ABB RobotStudio station: Session3b.rspag

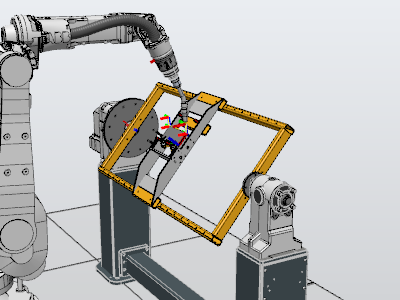
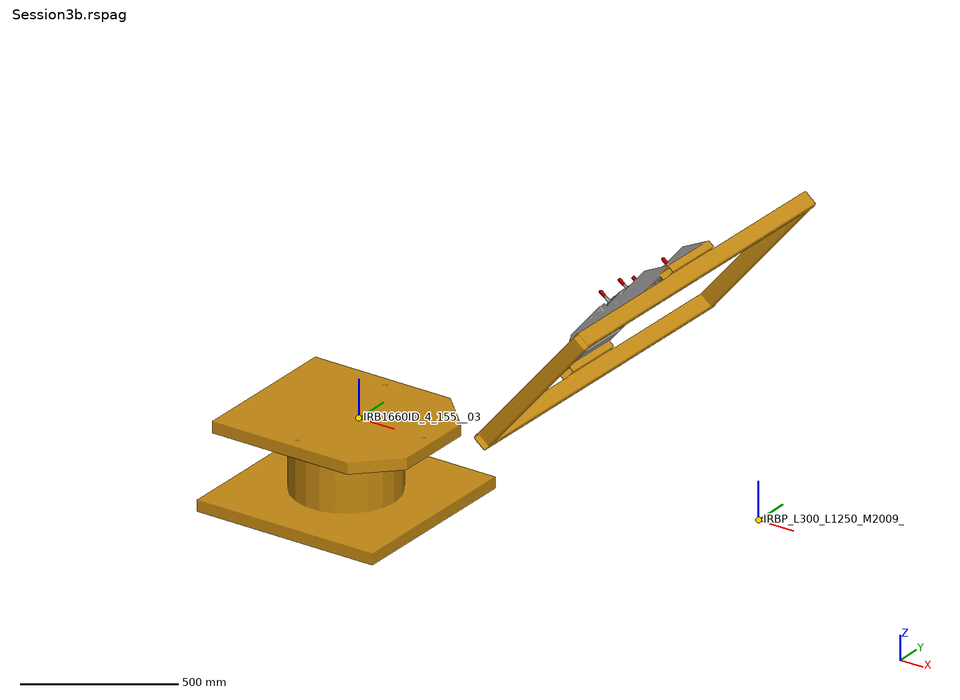
[picture v1: parts stored in the station drawn from their meshes, with robot base, taught points and paths (robot models come from the ABB library and are not in the file)]
--- station ---
Station Session3b (saved by RobotStudio 24.2.10821.1)
Controller Controller4, task T_ROB1: task frame (RAPID world) sits at (0, 0, 300) mm in the station
Controller Controller4
  mechanical unit ROB_1: IRB1660ID_4_155__03, 6 joints, base frame (0, 0, 0) mm
  mechanical unit STN1: IRBP_L300_L1250_M2009_REV1_01, 1 joints, base frame (1100, 625, 650) mm, rotated rx 0 ry -90 rz 90 deg
Layout (positions relative to the parent item):
  - IRB1660ID_4_155__03 [mechanism, from %ABB.RobotStudio.Models.IRB1660ID%\IRB1660ID_4_155__03.rslib] at (0, 0, 300) mm; joint values [-0.1022, 0.0725, -0.0812, 0.0517, 1.1108, -0.1141] (rad or m)
  - Binzel_ID_22 [mechanism, from %ABB.RobotStudio.Models.ArcWelding%\Binzel_ID_22.rslib] at (934.43, -89.58, 1480.22) mm, rotated rx -180 ry 27 rz -180 deg
  - IRBP_L300_L1250_M2009_REV1_01 [mechanism] at (1100, 625, 0) mm; joint values [0.8727] (rad or m)
      links: Base, Link1
  - test part [part] at (1100, 625, 950) mm, rotated rx -90 ry -40 rz 180 deg, size 190.1 x 652.8 x 1250 mm
  - robot stand [part], size 675 x 675 x 300 mm
Attachment: Binzel_ID_22 is attached to IRB1660ID_4_155__03 / Link6
Attachment: test part is attached to IRBP_L300_L1250_M2009_REV1_01 / Link1

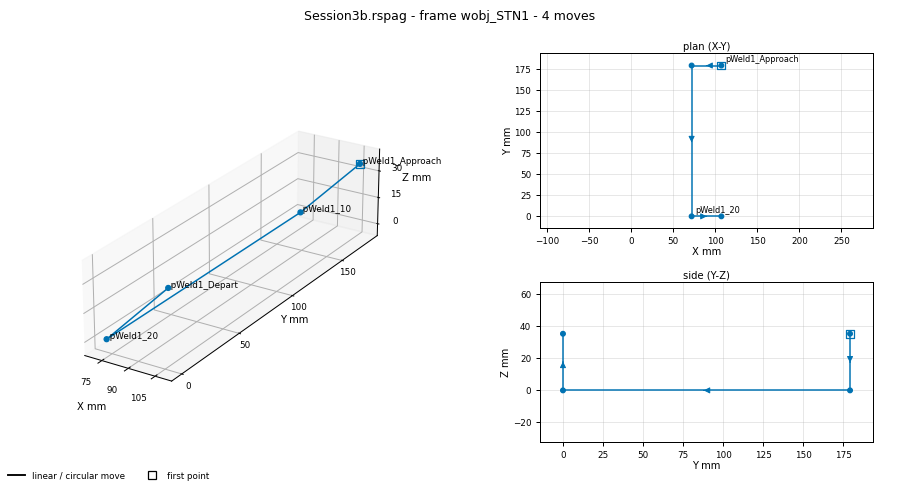
[picture p0: tool path of Session3b.rspag in frame wobj_STN1, 4 of 4 moves have a stored position in this frame; points joined in program order, loops and branches not executed]
--- Backups/Controller4/RAPID/TASK1/PROGMOD/CalibData.mod ---
MODULE CalibData
    PERS tooldata tWeldGun:=[TRUE,[[49.841566361,0,372.194826196],[0.981627183,0,0.190808995,0]],[2,[0,0,100],[0,1,0,0],0,0,0]];
    TASK PERS wobjdata wobj_STN1:=[FALSE,FALSE,"STN1",[[0,0,0],[1,0,0,0]],[[109.166,-1.08,714.579],[0.5,-0.5,0.5,-0.5]]];
ENDMODULE

--- Backups/Controller4/RAPID/TASK1/PROGMOD/Module1.mod ---
MODULE Module1
        CONST robtarget pWeld1_Approach:=[[107.355339022,179.2,35.355339096],[0.382683432,0,-0.923879533,0],[0,0,0,0],[9E+09,9E+09,9E+09,9E+09,45,9E+09]];
    CONST robtarget pWeld1_10:=[[72,179.2,0],[0.382683432,0,-0.923879533,0],[0,0,0,0],[9E+09,9E+09,9E+09,9E+09,60,9E+09]];
    CONST robtarget pWeld1_20:=[[72,0,0],[0.382683432,0,-0.923879533,0],[0,0,0,0],[9E+09,9E+09,9E+09,9E+09,80,9E+09]];
    CONST robtarget pWeld1_Depart:=[[107.355339022,0,35.355339096],[0.382683432,0,-0.923879533,0],[0,0,0,0],[9E+09,9E+09,9E+09,9E+09,50,9E+09]];
!***********************************************************
    !
    ! Module:  Module1
    !
    ! Description:
    !   <Insert description here>
    !
    ! Author: ahmadk
    !
    ! Version: 1.0
    !
    !***********************************************************


    !***********************************************************
    !
    ! Procedure main
    !
    !   This is the entry point of your program
    !
    !***********************************************************
    PROC main()
        !Add your code here
        Weld1;
    ENDPROC
    PROC Weld1()
        ActUnit STN1;
        MoveJ pWeld1_Approach,vmax,z10,tWeldGun\WObj:=wobj_STN1;
        MoveL pWeld1_10,v500,fine,tWeldGun\WObj:=wobj_STN1;
        MoveL pWeld1_20,v500,fine,tWeldGun\WObj:=wobj_STN1;
        MoveL pWeld1_Depart,v500,fine,tWeldGun\WObj:=wobj_STN1;
    ENDPROC
ENDMODULE

--- Backups/Controller4/SYSPAR/EIO.cfg ---
EIO:CFG_1.0:6:1::
#
LOCAL_DEVICE:

      -Name "DRVIO_1" -Network "Local" -StateWhenStartup "Deactivated"\
      -TrustLevel "DRVIO_TRUSTLEVEL"
#
EIO_CROSS:

      -Name "Cross_doACT_K1" -Res "doACT_K1" -Act1 "soACT_STN1"

      -Name "Cross_siSTN1_ACT" -Res "siSTN1_ACT" -Act1 "diK1_ACT"
#
EIO_DEVICE_TRUSTLEVEL:

      -Name "DRVIO_TRUSTLEVEL" -ActionWhenLost "NONE" -ReportWhenLost "NONE"\
      -ReportWhenReconnected "NONE"
#
EIO_SIGNAL:

      -Name "doACT_K1" -SignalType "DO" -Device "DRVIO_1" -DeviceMap "0"

      -Name "doACT_K11" -SignalType "DO" -Device "DRVIO_1" -DeviceMap "5"

      -Name "diK1_ACT" -SignalType "DI" -Device "DRVIO_1" -DeviceMap "0"\
      -FiltPas 50 -FiltAct 50

      -Name "soACT_STN1" -SignalType "DO" -DeviceMap "0"

      -Name "siSTN1_ACT" -SignalType "DI" -DeviceMap "0"
